// TwinCAT 3 PLC project Untitled1
// ProgramVersion: 3.1.4020.5
// libraries:
//   Tc2_Standard, * (Beckhoff Automation GmbH)
//   Tc2_System, * (Beckhoff Automation GmbH)
//   Tc3_Module, * (Beckhoff Automation GmbH)
// project tree:
//   DUTs/ DUT_ENUM_TEST.TcDUT, DUT_STRUCT_TEST.TcDUT
//   / PlcTask.TcTTO
//   POUs/ MAIN.TcPOU
// real-time tasks:
//   TASK PlcTask: cycle T#10ms, priority 20, ADS port 350

CONFIGURATION Untitled1
    RESOURCE PLC ON TwinCAT3
        TASK PlcTask(INTERVAL := T#10ms, PRIORITY := 20);
        PROGRAM MAIN WITH PlcTask : MAIN;
    END_RESOURCE
END_CONFIGURATION

// ---- DUTs/DUT_ENUM_TEST.TcDUT
{attribute 'qualified_only'}
{attribute 'strict'}
TYPE DUT_ENUM_TEST :
(
	zeroeth_member := 0,
	first_member := 1,
	second_member := 2,
	third_member := 3
);
END_TYPE

// ---- DUTs/DUT_STRUCT_TEST.TcDUT
TYPE DUT_STRUCT_TEST :
STRUCT

	{attribute 'pytmc' := '
		pv: ADS_TST:SetfAmpRB
		pv: ADS_TST:SetfAmp
		io: o
		pv: ADS_TST:GetfAmp
		io: i
	'}
	fAmplitude :	LREAL;
	{attribute 'pytmc' := '
		pv: ADS_TST:SetFArrayRB
		pv: ADS_TST:SetFArray
		io: o
		pv: ADS_TST:GetFArray
		io: i
	'}
	fArray : ARRAY [1..5] OF LREAL;
	{attribute 'pytmc' := '
		pv: ADS_TST:SetStrRB
		pv: ADS_TST:SetStr
		io: o
		pv: ADS_TST:GetStr
		io: i
	'}
	str	:	STRING(35);


END_STRUCT	
END_TYPE

// ---- POUs/MAIN.TcPOU
PROGRAM MAIN
VAR
	
	{attribute 'pytmc' := '
		pv: ADS_TST:SetiCycleRB
		pv: ADS_TST:SetiCycle
		io: o
		pv: ADS_TST:GetiCycle
		io: i
	'}
	iCycle : INT;

	{attribute 'pytmc' := '
		pv: ADS_TST:SetdiCycleRB
		pv: ADS_TST:SetdiCycle
		io: o
		pv: ADS_TST:GetdiCycle
		io: i
	'}
	diCycle : DINT;
	
	{attribute 'pytmc' := '
		pv: ADS_TST:SetbStateRB
		pv: ADS_TST:SetbState
		io: o
		pv: ADS_TST:GetbState
		io: i
	'}
	bState : BOOL;

	{attribute 'pytmc' := '
		pv: ADS_TST:SetlrAmpRB
		pv: ADS_TST:SetlrAmp
		io: o
		pv: ADS_TST:GetlrAmp
		io: i
	'}
	lrAmplitude :	LREAL;

	{attribute 'pytmc' := '
		pv: ADS_TST:SetrAmpRB
		pv: ADS_TST:SetrAmp
		io: o
		pv: ADS_TST:GetrAmp
		io: i
	'}
	rAmplitude :	REAL;

	{attribute 'pytmc' := '
		pv: ADS_TST:SetlrArrayRB
		pv: ADS_TST:SetlrArray
		io: o
		pv: ADS_TST:GetlrArray
		io: i
	'}
	lrArray : ARRAY [1..5] OF LREAL;

	{attribute 'pytmc' := '
		pv: ADS_TST:SetrArrayRB
		pv: ADS_TST:SetrArray
		io: o
		pv: ADS_TST:GetrArray
		io: i
	'}	
	rArray : ARRAY [1..5] OF REAL;

	{attribute 'pytmc' := '
		pv: ADS_TST:SetiArrayRB
		pv: ADS_TST:SetiArray
		io: o
		pv: ADS_TST:GetiArray
		io: i
	'}
	iArray : ARRAY [1..5] OF INT;

	{attribute 'pytmc' := '
		pv: ADS_TST:SetdiArrayRB
		pv: ADS_TST:SetdiArray
		io: o
		pv: ADS_TST:GetrdiArray
		io: i
	'}
	diArray : ARRAY [1..5] OF DINT;
	
	
	{attribute 'pytmc' := '
		pv: ADS_TST:SetbArrayRB
		pv: ADS_TST:SetbArray
		io: o
		pv: ADS_TST:GetbArray
		io: i
	'}
	bArray : ARRAY [1..5] OF BOOL;
	
	is_true : BOOL;
	is_false : BOOL;
	val : BOOL;
	dval : DINT;

	{attribute 'pytmc' := '
		pv: ADS_TST:SetStrRB
		pv: ADS_TST:SetStr
		io: o
		pv: ADS_TST:GetStr
		io: i
	'}
	sTest	:	STRING(35);
	
	
	
	{attribute 'pytmc' := '
		pv: ADS_TST:SeteStatusRB
		pv: ADS_TST:SeteStatus
		io: o
		pv: ADS_TST:GeteStatus
		io: i
	'}	
	eStatus	:	DUT_ENUM_TEST;

	{attribute 'pytmc' := '
		pv: ADS_TST:SetenumArrayRB
		pv: ADS_TST:SetenumArray
		io: o
		pv: ADS_TST:GetenumArray
		io: i
	'}	
	enumArray	: ARRAY [1..5] of DUT_ENUM_TEST;



	
	{attribute 'pytmc' := '
		pv: ADS_TST:SetStrRB
	'}
	//structure_type : DUT_STRUCT_TEST;
	
	// *****************************
	//bool_type : BOOL;
	
	//enum_type : DUT_ENUM_TEST; 
END_VAR

IF bArray[1] = TRUE THEN
	is_true := TRUE;
	is_false := FALSE;

else
	is_true := FALSE;
	is_false := TRUE;
END_IF


val := bArray[1];

END_PROGRAM
